FUNCTION_BLOCK POU
VAR_IN_OUT
	out : ARRAY[*] OF BOOL;
END_VAR
VAR
	timer : TON;
	i : DINT;
END_VAR

IF i > UPPER_BOUND(out, 1) THEN
	RETURN;
END_IF

IF i = LOWER_BOUND(out, 1) THEN //if first ouptut does not need delay
	out[i] := TRUE;
	i := i + 1;
	RETURN;
END_IF


timer(IN:= , PT:= T#1S, Q=> out[i], ET=> );
timer.IN := TRUE;
IF timer.Q THEN
	//out[i-1] := FALSE; //turn off previous output, optional
	i := i + 1;
	timer.IN := FALSE;
END_IF

END_FUNCTION_BLOCK

(* stored: Version 1.1.0.1, ProductVersion 3.1.4024.11
   POU POU: Id {8b206f4b-01bb-4bf9-a81f-4c6ae99f8f28}, SpecialFunc None *)
